TYPE ST_System_MVHW_Stellwert :
STRUCT
	Anford_Stellventil		: BOOL;
	Anford_Pumpe		: BOOL;
	Anford_Kompressor	: BOOL;
END_STRUCT
END_TYPE

(* stored: Version 1.1.0.1, ProductVersion 3.1.4024.9
   DUT ST_System_MVHW_Stellwert: Id {c5445bae-375b-44fd-97d6-d526c8ee52e0} *)
